Fanuc KAREL source: kt00406.KL

-- PROVISIONAL review KL for V770-1; original PC SHA256 9830fcf1d715f839cb45bbdf3bbc18f3abdf8ce918aa384c3aed64ee7417c91e
-- Incomplete behavior may be omitted. Consult companion uncertainty JSON. Do not deploy.
PROGRAM KT00406
%NOLOCKGROUP
VAR
  R1 : REAL
  R2 : REAL
  OUT : BOOLEAN
BEGIN
  -- UNRESOLVED_PC offsets 5-16; opcodes 2E,23
  -- UNRESOLVED_PC offsets 21-32; opcodes 2E,23
  -- UNRESOLVED_PC offsets 37-48; opcodes 2E,23
  -- UNRESOLVED_PC offsets 53-64; opcodes 2E,23
  -- UNRESOLVED_PC offsets 69-88; opcodes 21,21,71,23
  -- UNRESOLVED_PC offsets 93-97; opcodes 7F
END KT00406
